{attribute addProperty BoxType "EL3773-0000-0016"}
{attribute addProperty Id "Cycle_CountAT %I*UINT162"}
{attribute addProperty CRC "2363401108"}
{attribute addProperty SizeInBites "16"}
{attribute addProperty SizeInBytes "2"}
TYPE AI_CycleCount_8CDEA394 :
STRUCT
	{attribute addProperty Name "Cycle_Count"}
	Cycle_Count AT %I* : UINT;
END_STRUCT
END_TYPE

(* stored: Version 1.2.0.0, ProductVersion 3.1.4024.9
   DUT AI_CycleCount_8CDEA394: Id {5f76c994-db3c-44da-9cf1-e54593077ae4} *)
